// TIA Portal V19 export
FUNCTION_BLOCK "Temperature Type"   // FB4, LAD
{ S7_Optimized_Access := 'TRUE' }
// stored: MemoryReserve 100, SetENOAutomatically false
   VAR_INPUT
      "RAW INPUT" : Int;
      "Scale MIN" : Real;
      "Scale MAX" : Real;
   END_VAR
   VAR_OUTPUT
      PV : Real;
   END_VAR
   VAR
      IEC_Timer_0_Instance_2 { S7_SetPoint := 'True'} : TON_TIME;
      IEC_Timer_0_Instance { S7_SetPoint := 'True'} : TOF_TIME;
      "INT TO REAL" : Real;
   END_VAR
   VAR CONSTANT
      "0" : Int := 0;
      "1" : Int := 1;
   END_VAR
BEGIN

REGION Network 1
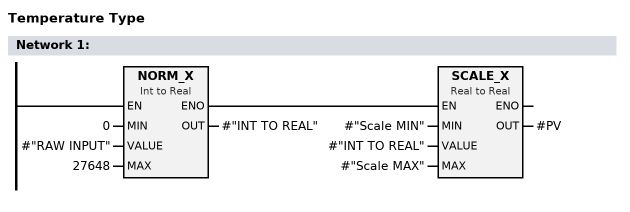
   RUNG wire#powerrail
      { S7_Templates := "[SrcType := Int, DestType := Real]" } Normalize(min := 0, value := #"RAW INPUT", max := 27648, out => #"INT TO REAL")
      { S7_Templates := "[SrcType := Real, DestType := Real]" } Scale(min := #"Scale MIN", value := #"INT TO REAL", max := #"Scale MAX", out => #PV)
   END_RUNG
   // the same network as SCL:
   #"INT TO REAL" := NORM_X(MIN := 0, VALUE := #"RAW INPUT", MAX := 27648);
   #PV := SCALE_X(MIN := #"Scale MIN", VALUE := #"INT TO REAL", MAX := #"Scale MAX");
END_REGION
END_FUNCTION_BLOCK
